FUNCTION Convert_DATE_TO_DATE : Hresult
VAR_INPUT
	in : DATE;
	out : REFERENCE TO DATE;
END_VAR

out := in;

END_FUNCTION

(* stored: Version 1.1.0.1, ProductVersion 3.1.4024.12
   POU Convert_DATE_TO_DATE: Id {7116e533-ce53-4987-a18b-0d0381f360a2}, SpecialFunc None *)
